FUNCTION F_TemperatureMonitor_Error : FB_TemperatureMonitor
VAR_INPUT
END_VAR
VAR_OUTPUT
	stSetpoints : ST_TemperatureMonitorSetpoints := F_TemperatureMonitorSetpoints();
END_VAR
VAR
	fbTempMon : FB_TemperatureMonitor;
END_VAR

fbTempMon(
	nTempMonRaw := 16#7736,
	bAmphosOn := TRUE,
	stSetpoints := stSetpoints
);
F_TemperatureMonitor_Error := fbTempMon;

END_FUNCTION

(* stored: Version 1.1.0.1, ProductVersion 3.1.4020.14
   POU F_TemperatureMonitor_Error: Id {ef28fab8-7efb-4999-980f-8b5e3f6f9379}, SpecialFunc None *)
